FUNCTION_BLOCK TEST_ABS (* Test absolute value functions *)
  (* Standard: 61499-2 *)
  (* Version 0.0, 2006-09-02, JHC, Holobloc Inc *)
  (* Compiler header: package fb.rt.test; *)
  (* Compiler classdef: SimpleFB *)
  (* Compiler Java Sun JDK 1.5.0 *)
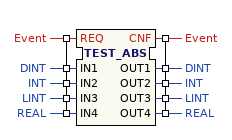
  EVENT_INPUT
    REQ WITH IN1, IN2, IN3, IN4; (* Normal Execution Request *)
  END_EVENT
  EVENT_OUTPUT
    CNF WITH OUT1, OUT2, OUT3, OUT4; (* Execution Confirmation *)
  END_EVENT
  VAR_INPUT
    IN1 : DINT;
    IN2 : INT;
    IN3 : LINT;
    IN4 : REAL;
  END_VAR
  VAR_OUTPUT
    OUT1 : DINT;
    OUT2 : INT;
    OUT3 : LINT;
    OUT4 : REAL;
  END_VAR
  ALGORITHM REQ IN FBD: (* Normally executed algorithm *)
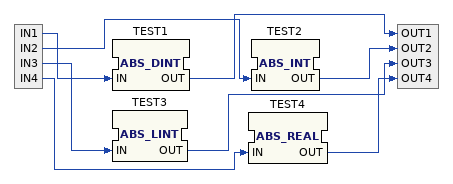
    FBS
      TEST1 : ABS_DINT;
      TEST2 : ABS_INT;
      TEST3 : ABS_LINT;
      TEST4 : ABS_REAL;
    END_FBS
    DATA_CONNECTIONS
      IN1 TO TEST1.IN;
      IN2 TO TEST2.IN;
      IN3 TO TEST3.IN;
      IN4 TO TEST4.IN;
      TEST1.OUT TO OUT1;
      TEST2.OUT TO OUT2;
      TEST3.OUT TO OUT3;
      TEST4.OUT TO OUT4;
    END_CONNECTIONS
  END_ALGORITHM
END_FUNCTION_BLOCK
